// TIA Portal V18 export
// export: Created 2025-12-01T12:38:07.0590817Z, ExportSetting None, DisplayName Totally Integrated Automation Portal, DisplayVersion V18 Update 5, DisplayName TIA Portal Openness, DisplayVersion V18 Update 5, DisplayName TIA Portal Teamcenter Gateway, DisplayVersion V18, DisplayName TIA Portal Version Control Interface, DisplayVersion V18, DisplayName STEP 7 Professional, DisplayVersion V18 Update 5, DisplayName STEP 7 Safety, DisplayVersion V18, DisplayName WinCC Professional, DisplayVersion V18 Update 5
DATA_BLOCK "AutoProcessData"   // DB1600
{ S7_Optimized_Access := 'FALSE' }
// stored: AutoNumber false
   VAR RETAIN
      A_ScanRotate : "ProcessData";
      F_Robot1Grip1 { S7_SetPoint := 'True'} : "ProcessData";
      F_Robot1Grip2 { S7_SetPoint := 'True'} : "ProcessData";
      B_Press1 { S7_SetPoint := 'True'} : "ProcessData";
      C_Glue { S7_SetPoint := 'True'} : "ProcessData";
      F_Robot2Grip1 { S7_SetPoint := 'True'} : "ProcessData";
      F_Robot2Grip2 { S7_SetPoint := 'True'} : "ProcessData";
      C_GlueNGBuffer { S7_SetPoint := 'True'} : "ProcessData";
      C_MagnScanNGBuffer { S7_SetPoint := 'True'} : "ProcessData";
      B_Press2 { S7_SetPoint := 'True'} : "ProcessData";
      F_Robot3Grip1 { S7_SetPoint := 'True'} : "ProcessData";
      F_Robot3Grip2 { S7_SetPoint := 'True'} : "ProcessData";
      H_ShafeLine { S7_SetPoint := 'True'} : "ProcessData";
      J_ShafeLine { S7_SetPoint := 'True'} : "ProcessData";
      K_ShafeLine { S7_SetPoint := 'True'} : "ProcessData";
      L_ShafeLine { S7_SetPoint := 'True'} : "ProcessData";
      ClearData { S7_SetPoint := 'True'} : "ProcessData";
      A_Table_1 { S7_SetPoint := 'True'} : Array[1..10] of "TableProcessData";
      A_Table_2 { S7_SetPoint := 'True'} : Array[1..10] of "TableProcessData";
      FixtureCode_A1 { S7_SetPoint := 'True'} : Array[1..10] of String[128];
      FixtureCode_A2 { S7_SetPoint := 'True'} : Array[1..10] of String[128];
      GlobalData : Struct
         Table1CodeOKFlag : Bool;
         Table2CodeOKFlag : Bool;
         Fixture1CodeOKFlag : Bool;
         Fixture2CodeOKFlag : Bool;
         Robot2GripperCodeOKFlag : Bool;
         Robot1GripperCodeOKFlag : Bool;
         Robot3GripperCodeOKFlag : Bool;
         Spare_8 : Bool;
         Spare_9 : Bool;
         Spare_10 : Bool;
         Spare_11 : Bool;
         Spare_12 : Bool;
         Spare_13 : Bool;
         Spare_14 : Bool;
         Spare_15 : Bool;
         Spare_16 : Bool;
         DataIndex { S7_SetPoint := 'True'} : Int := 1;
         Robot1GripCodeStatus1 : Int;
         Robot1GripCodeStatus2 : Int;
         Robot1GripCodeStatus3 : Int;
         Robot1GripCodeStatus4 : Int;
         Robot2GripCodeStatus1 : Int;
         Robot2GripCodeStatus2 : Int;
         Robot2GripCodeStatus3 : Int;
         Robot2GripCodeStatus4 : Int;
         Robot3GripCodeStatus1 : Int;
         Robot3GripCodeStatus2 : Int;
         Robot3GripCodeStatus3 : Int;
         Robot3GripCodeStatus4 : Int;
         FixtureCode_A1Status1 : Int;
         FixtureCode_A1Status2 : Int;
         FixtureCode_A1Status3 : Int;
         FixtureCode_A1Status4 : Int;
         FixtureCode_A1Status5 : Int;
         FixtureCode_A1Status6 : Int;
         FixtureCode_A1Status7 : Int;
         FixtureCode_A1Status8 : Int;
         FixtureCode_A1Status9 : Int;
         FixtureCode_A1Status10 : Int;
         FixtureCode_A2Status1 : Int;
         FixtureCode_A2Status2 : Int;
         FixtureCode_A2Status3 : Int;
         FixtureCode_A2Status4 : Int;
         FixtureCode_A2Status5 : Int;
         FixtureCode_A2Status6 : Int;
         FixtureCode_A2Status7 : Int;
         FixtureCode_A2Status8 : Int;
         FixtureCode_A2Status9 : Int;
         FixtureCode_A2Status10 : Int;
         Spare : Array[1..332] of Byte;
      END_STRUCT;
      DataBuffer : Array[1..30] of "ProcessData";
      GripperCode_R1 { S7_SetPoint := 'True'} : Array[1..10] of String[128];
      GripperCode_R2 { S7_SetPoint := 'True'} : Array[1..10] of String[128];
      GripperCode_R3 { S7_SetPoint := 'True'} : Array[1..10] of String[128];
   END_VAR
BEGIN
   A_Table_1[1].Code := 'SZ23055-OP010-E-Compressor-ring1 Loading tooling-1';
   A_Table_1[2].Code := 'SZ23055-OP010-E-Compressor-ring1 Loading tooling-2';
   A_Table_2[1].Code := 'SZ23055-OP010-E-Compressor-ring2 Loading tooling-1$R';
END_DATA_BLOCK
